Fanuc KAREL source: kt00084.KL

-- PROVISIONAL review KL for V770-1; original PC SHA256 f712eeef60d52e70e1824e359377fcd880f0744bda7f370b4f760ed61ec2829b
-- Incomplete behavior may be omitted. Consult companion uncertainty JSON. Do not deploy.
PROGRAM KT00084
%NOLOCKGROUP
VAR
  R2 : REAL
  OUT : REAL
-- UNRESOLVED_DECL Y1 type=002018
BEGIN
  -- UNRESOLVED_PC offsets 5-19; opcodes 2E,22,9D,33,B2
  -- UNRESOLVED_PC offsets 24-35; opcodes 2E,23
  -- UNRESOLVED_PC offsets 40-64; opcodes 22,9D,33,B1,21,29,64,6B,23
  -- UNRESOLVED_PC offsets 69-73; opcodes 7F
END KT00084
